Fanuc KAREL source: kt00896.KL

-- PROVISIONAL review KL for V940-1; original PC SHA256 df791889ee46ce3673a1073115cf94ffe0c9dd5444f8089a8047f15d1a96ef36
-- Incomplete behavior may be omitted. Consult companion uncertainty JSON. Do not deploy.
PROGRAM KT00896
%NOLOCKGROUP
VAR
  OUT : BOOLEAN
-- UNRESOLVED_DECL P1 type=000199
-- UNRESOLVED_DECL P2 type=000199
BEGIN
  -- V9_ZERO_TABLE_METADATA_HINT layout=0001; no indexed target words; source/name/runtime held
  -- UNRESOLVED_PC offsets 5-31; opcodes 27,27,49,7E,AD,27,9D,76,23
  -- UNRESOLVED_PC offsets 36-40; opcodes 7F
END KT00896
